(* CoDeSys 2.3 export: CreateGlobalBufferHandle.EXP *)

(* POU basic/CreateGlobalBufferHandle, ST *)
FUNCTION CreateGlobalBufferHandle : BOOL
VAR_INPUT
    BufferAddress: DWORD;
    BufferSize: DINT;
END_VAR
VAR
END_VAR
CreateBufferHandle(BufferAddress, BufferSize, GlobalLogBufferHandle);
END_FUNCTION
